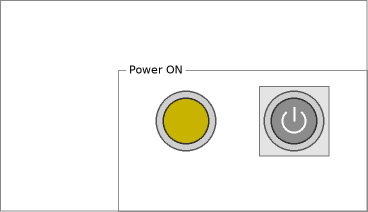
VISUALIZATION Visualization  // 368x212
    GroupBox (118,62 250x150), "Power ON"
        Lamp1 (33,24 70x70), style: Lamp-Lamp1-Yellow
        PowerSwitch (141,24 70x70), behaviour: TOGGLE, style: Switch-PowerSwitch-Gray
END_VISUALIZATION

(* stored: Version 1.1.0.1, ProductVersion 3.1.4024.12
   Visu Visualization: Id {e33c69bc-1615-43bf-91d8-f6e34270db4d} *)
